Staubli VAL3: Body.pjx

--- Body.pjx ---
Parameters version=s7.7.2 stackSize=5000 millimeterUnit=true
Program file=start.pgx
Program file=stop.pgx
Data file=Body.dtx

--- Body.dtx ---
mdesc mNomSpeed
public num nData
